Fanuc TP program (LS listing): _set_wait.ls

/PROG  _SET_WAIT
/ATTR
OWNER		= MNEDITOR;
COMMENT		= "Set-WAITTMOUT";
PROG_SIZE	= 378;
CREATE		= DATE 22-04-05  TIME 09:41:30;
MODIFIED	= DATE 26-06-29  TIME 14:54:08;
FILE_NAME	= ;
VERSION		= 0;
LINE_COUNT	= 9;
MEMORY_SIZE	= 746;
PROTECT		= READ_WRITE;
TCD:  STACK_SIZE	= 0,
      TASK_PRIORITY	= 50,
      TIME_SLICE	= 0,
      BUSY_LAMP_OFF	= 0,
      ABORT_REQUEST	= 0,
      PAUSE_REQUEST	= 0;
DEFAULT_GROUP	= 1,*,*,*,*;
CONTROL_CODE	= 00000000 00000000;
LOCAL_REGISTERS	= 0,0,0;
/MN
   1:  $SSR.$STEPSTMTTYP=1 ;
   2:  !*****SET WAIT-TIMEOUT TIME****** ;
   3:  R[391:*Timeout-Set]=AR[1]    ;
   4:  IF (R[391:*Timeout-Set]=0) THEN ;
   5:  $WAITTMOUT=R[390:Timeout-Def] ;
   6:  ELSE ;
   7:  $WAITTMOUT=R[391:*Timeout-Set] ;
   8:  ENDIF ;
   9:  $SSR.$STEPSTMTTYP=3 ;
/POS
/END
